{attribute 'reflection'}
FUNCTION_BLOCK ACObject IMPLEMENTS IACObject
VAR_INPUT
END_VAR
VAR_OUTPUT
	_InstanceID : UDINT;
	{attribute 'instance-path'}
	{attribute 'no_init'}
	_ACUrl : STRING(GCL.cACUrlLEN);
END_VAR
VAR
	_FBInitCount : UDINT;
	_MaxPropertyID : UINT;
END_VAR

PROPERTY ACInitState : ACInitStateEnum
GET
IF _InstanceID = 0 OR _FBInitCount = 0 THEN
	ACInitState := ACInitStateEnum.NewInstance;
	RETURN;
ELSIF NOT (_InstanceID = _FBInitCount) THEN
	ACInitState := ACInitStateEnum.Reinitialized;
	RETURN;
END_IF
ACInitState := ACInitStateEnum.Unchanged;
END_GET
END_PROPERTY

{attribute 'TcRpcEnable'}
PROPERTY ACUrl : STRING
GET
ACUrl := _ACUrl;
END_GET
END_PROPERTY

// Short ACUrl Without ".PLC.MAIN"-Prefix
PROPERTY ACUrlS : STRING
GET
VAR
	pos: INT;
END_VAR
IF LEN(_ACUrl) = 0 THEN
	ACUrlS := _ACUrl;
	RETURN;
END_IF

pos := FIND(_ACUrl,GCL.cPathMAIN);
IF pos <= 0 THEN
	ACUrlS := _ACUrl;
	RETURN;
END_IF

ACUrlS := RIGHT(_ACUrl,LEN(_ACUrl) - pos-LEN(GCL.cPathMAIN)+1);
END_GET
END_PROPERTY

METHOD FB_postinit
VAR_INPUT
	root : IACVariobatch;
END_VAR
GVL.gInstanceIDCount := GVL.gInstanceIDCount + 1;
_InstanceID := GVL.gInstanceIDCount;
_FBInitCount := _InstanceID;
_MaxPropertyID := 0;
root.SetCompMetadata(THIS^);
OnInitMemory(root);
END_METHOD

METHOD FindObjectInChilds : IACObject
VAR_INPUT
	instanceID	: UDINT;
END_VAR
FindObjectInChilds := 0;
END_METHOD

METHOD PROTECTED IncFBInitCount
VAR_INPUT
END_VAR
GVL.gFBInitCount := GVL.gFBInitCount + 1;
_FBInitCount := GVL.gFBInitCount;
GVL.gInstanceIDCount := 0;
END_METHOD

{attribute 'TcRpcEnable'}
PROPERTY InstanceID : UDINT
GET
InstanceID := _InstanceID;
END_GET
END_PROPERTY

PROPERTY MaxPropertyID : UINT
GET
MaxPropertyID := _MaxPropertyID;
END_GET
END_PROPERTY

METHOD OnInitMemory
VAR_INPUT
		root : IACVariobatch;
END_VAR
root.OnObjectMetaBuilded(THIS^);
END_METHOD

METHOD RegisterProperty
VAR_INPUT
	root : IACVariobatch;
	propertyID : UINT;
	sizeOfPropType : WORD;
END_VAR
IF propertyID > _MaxPropertyID THEN
	_MaxPropertyID := propertyID;
END_IF
root.SetPropMetadata(THIS^,propertyID,sizeOfPropType);
END_METHOD

{attribute 'TcRpcEnable'}
PROPERTY ThisPointer : LWORD
GET
ThisPointer := THIS;
END_GET
END_PROPERTY

PROPERTY PUBLIC TypeOfACObject : TypeOfACObjectEnum
GET
TypeOfACObject := TypeOfACObjectEnum.Unknown;
END_GET
END_PROPERTY

END_FUNCTION_BLOCK

(* stored: Version 1.1.0.1, ProductVersion 3.1.4024.6
   POU ACObject: Id {6f57e18e-3f0d-41bf-b3e5-c82e8055ecf4}, SpecialFunc None
   Property ACInitState: Id {0492bcb1-381f-4689-8c6b-27011c1ceff8}
   Get Get: Id {b43b107b-a444-4c85-90e3-1e65840a4f92}
   Property ACUrl: Id {69197c2c-b889-4e00-bb7c-e34f6d789088}
   Get Get: Id {bb95567f-23ae-45bc-81b0-44e15c808f34}
   Property ACUrlS: Id {72b389be-6791-477d-96c0-a08130fccfa9}
   Get Get: Id {1ed57820-67c4-4456-b28c-1c84d681b3db}
   Method FB_postinit: Id {d6036f21-587f-460c-83a8-ab798ca9b231}
   Method FindObjectInChilds: Id {8e13438a-c304-416a-8e9c-3a30f15f5ccf}
   Method IncFBInitCount: Id {edb8ffb5-dc51-4fd2-9821-cce62dc2286a}
   Property InstanceID: Id {747db777-6d94-413f-8525-2b45eb89495f}
   Get Get: Id {5b764f71-600e-4a85-947c-48cb2c2cf98f}
   Property MaxPropertyID: Id {57eaefa8-406c-4d1c-b1a5-df160a5e78d7}
   Get Get: Id {c2dc703d-fe4e-407c-9ec7-e011a170b2c8}
   Method OnInitMemory: Id {5719f8c0-6380-433b-9d7b-650a01930144}
   Method RegisterProperty: Id {c9e67df5-3d56-4f21-86f3-30a025b57daf}
   Property ThisPointer: Id {54a94722-f531-4710-a4a5-c1b244504d20}
   Get Get: Id {c3957a32-30e4-4160-8b58-a3e3061ec547}
   Property TypeOfACObject: Id {8ae2ede3-a174-4731-9f69-1fd56baa4134}
   Get Get: Id {a6e3689f-4e18-4432-9fe1-d30d4b4e22b4} *)
